FUNCTION_BLOCK Globales_monolitico
VAR_INPUT
END_VAR
VAR_OUTPUT
END_VAR
VAR
END_VAR

END_FUNCTION_BLOCK

(* stored: Version 1.1.0.1, ProductVersion 3.1.4024.11
   POU Globales_monolitico: Id {cdd81dfd-df97-4b3b-b674-a3aed90a8356}, SpecialFunc None *)
